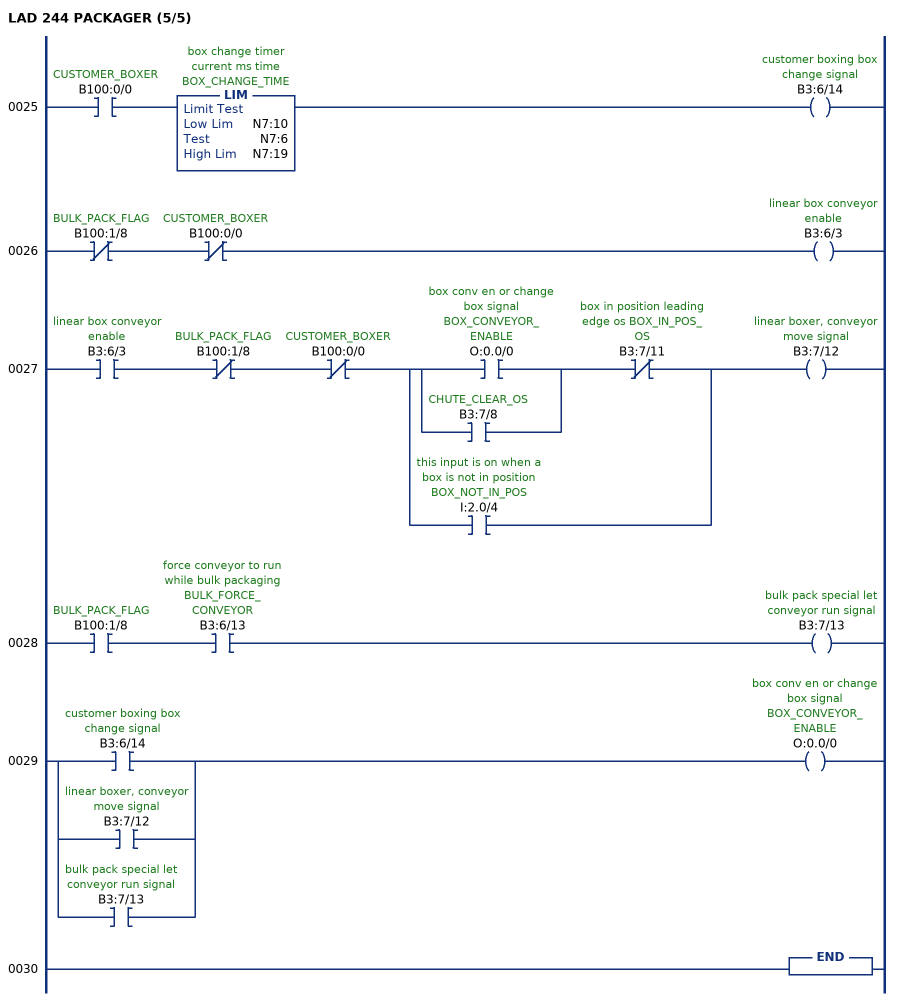
% Rung: 25 %
SOR XIC B100:0/0 LIM N7:10 N7:6 N7:19 OTE B3:6/14 EOR
%   B100:0/0  CUSTOMER_BOXER %
%   N7:10  CHUTE_CLOSED_TIME  "time at which chute door is considered closed" %
%   N7:6  BOX_CHANGE_TIME  "box change timer current ms time" %
%   N7:19  "end of customer boxer, box change signal" %
%   B3:6/14  "customer boxing box change signal" %
% Rung: 26 %
SOR XIO B100:1/8 XIO B100:0/0 OTE B3:6/3 EOR
%   B100:1/8  BULK_PACK_FLAG %
%   B100:0/0  CUSTOMER_BOXER %
%   B3:6/3  "linear box conveyor enable" %
% Rung: 27 %
SOR XIC B3:6/3 XIO B100:1/8 XIO B100:0/0 BST BST XIC O:0.0/0 NXB XIC B3:7/8 BND XIO B3:7/11 NXB XIC I:2.0/4 BND OTE B3:7/12 EOR
%   B3:6/3  "linear box conveyor enable" %
%   B100:1/8  BULK_PACK_FLAG %
%   B100:0/0  CUSTOMER_BOXER %
%   O:0.0/0  BOX_CONVEYOR_ENABLE  "box conv en or change box signal" %
%   B3:7/8  CHUTE_CLEAR_OS %
%   B3:7/11  BOX_IN_POS_OS  "box in position leading edge os" %
%   I:2.0/4  BOX_NOT_IN_POS  "this input is on when a box is not in position" %
%   B3:7/12  "linear boxer, conveyor move signal" %
% Rung: 28 %
SOR XIC B100:1/8 XIC B3:6/13 OTE B3:7/13 EOR
%   B100:1/8  BULK_PACK_FLAG %
%   B3:6/13  BULK_FORCE_CONVEYOR  "force conveyor to run while bulk packaging" %
%   B3:7/13  "bulk pack special let conveyor run signal" %
% Rung: 29 %
SOR BST XIC B3:6/14 NXB XIC B3:7/12 NXB XIC B3:7/13 BND OTE O:0.0/0 EOR
%   B3:6/14  "customer boxing box change signal" %
%   B3:7/12  "linear boxer, conveyor move signal" %
%   B3:7/13  "bulk pack special let conveyor run signal" %
%   O:0.0/0  BOX_CONVEYOR_ENABLE  "box conv en or change box signal" %
% Rung: 30 %
SOR END EOR

LADDER 245 "NO PACKAGE"
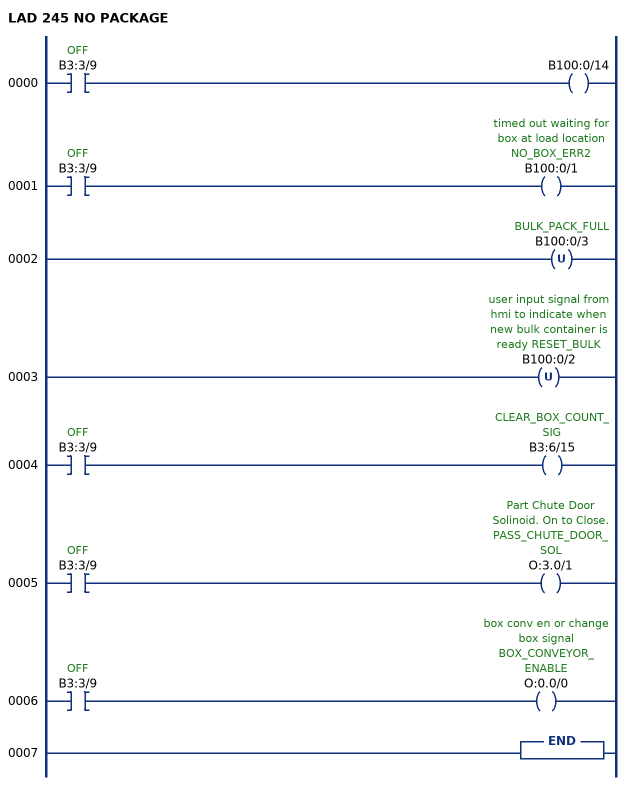
% Rung: 0 %
SOR XIC B3:3/9 OTE B100:0/14 EOR
%   B3:3/9  OFF %
% Rung: 1 %
SOR XIC B3:3/9 OTE B100:0/1 EOR
%   B3:3/9  OFF %
%   B100:0/1  NO_BOX_ERR2  "timed out waiting for box at load location" %
% Rung: 2 %
SOR OTU B100:0/3 EOR
%   B100:0/3  BULK_PACK_FULL %
% Rung: 3 %
SOR OTU B100:0/2 EOR
%   B100:0/2  RESET_BULK  "user input signal from hmi to indicate when new bulk container is ready" %
% Rung: 4 %
SOR XIC B3:3/9 OTE B3:6/15 EOR
%   B3:3/9  OFF %
%   B3:6/15  CLEAR_BOX_COUNT_SIG %
% Rung: 5 %
SOR XIC B3:3/9 OTE O:3.0/1 EOR
%   B3:3/9  OFF %
%   O:3.0/1  PASS_CHUTE_DOOR_SOL  "Part Chute Door Solinoid. On to Close." %
% Rung: 6 %
SOR XIC B3:3/9 OTE O:0.0/0 EOR
%   B3:3/9  OFF %
%   O:0.0/0  BOX_CONVEYOR_ENABLE  "box conv en or change box signal" %
% Rung: 7 %
SOR END EOR

LADDER 246 "RATE1"
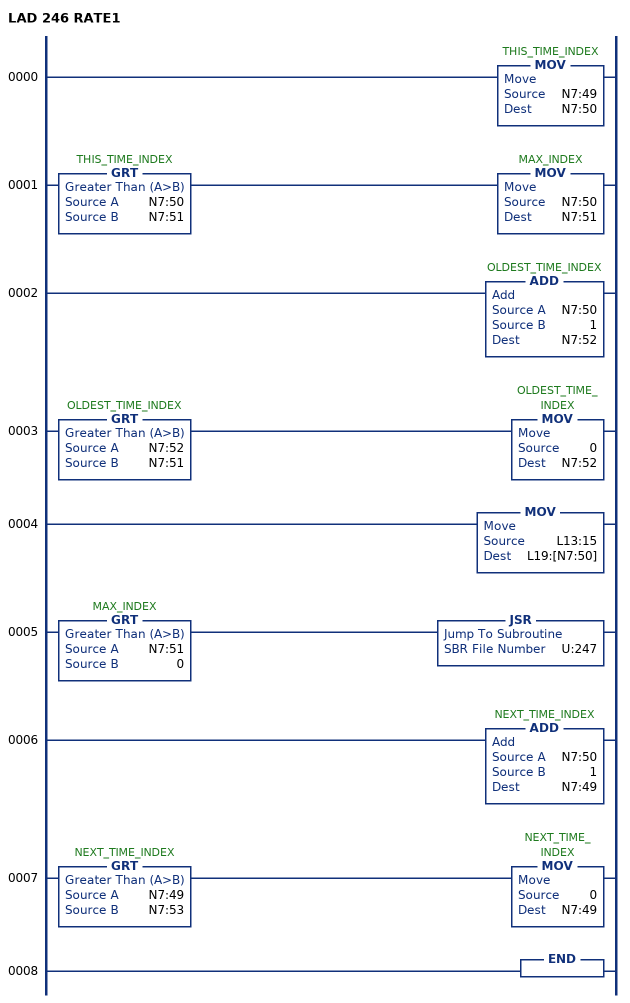
% Rung: 0 %
SOR MOV N7:49 N7:50 EOR
%   N7:49  NEXT_TIME_INDEX %
%   N7:50  THIS_TIME_INDEX %
% Rung: 1 %
SOR GRT N7:50 N7:51 MOV N7:50 N7:51 EOR
%   N7:50  THIS_TIME_INDEX %
%   N7:51  MAX_INDEX %
% Rung: 2 %
SOR ADD N7:50 1 N7:52 EOR
%   N7:50  THIS_TIME_INDEX %
%   N7:52  OLDEST_TIME_INDEX %
% Rung: 3 %
SOR GRT N7:52 N7:51 MOV 0 N7:52 EOR
%   N7:52  OLDEST_TIME_INDEX %
%   N7:51  MAX_INDEX %
% Rung: 4 %
SOR MOV L13:15 L19:[N7:50] EOR
%   L13:15  THE_TIME %
%   N7:50  THIS_TIME_INDEX %
% Rung: 5 %
SOR GRT N7:51 0 JSR U:247 EOR
%   N7:51  MAX_INDEX %
% Rung: 6 %
SOR ADD N7:50 1 N7:49 EOR
%   N7:50  THIS_TIME_INDEX %
%   N7:49  NEXT_TIME_INDEX %
% Rung: 7 %
SOR GRT N7:49 N7:53 MOV 0 N7:49 EOR
%   N7:49  NEXT_TIME_INDEX %
%   N7:53  UPPER_INDEX_LIMIT %
% Rung: 8 %
SOR END EOR

LADDER 247 "RATE2"
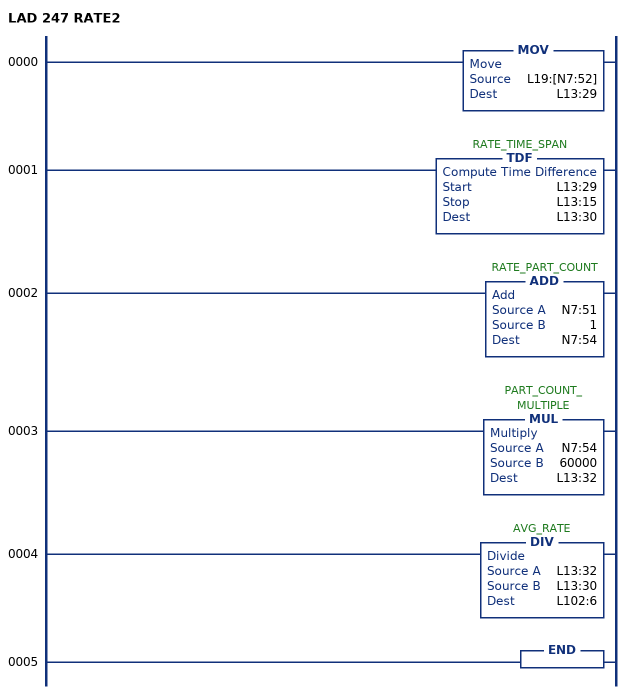
% Rung: 0 %
SOR MOV L19:[N7:52] L13:29 EOR
%   N7:52  OLDEST_TIME_INDEX %
% Rung: 1 %
SOR TDF L13:29 L13:15 L13:30 EOR
%   L13:15  THE_TIME %
%   L13:30  RATE_TIME_SPAN %
% Rung: 2 %
SOR ADD N7:51 1 N7:54 EOR
%   N7:51  MAX_INDEX %
%   N7:54  RATE_PART_COUNT %
% Rung: 3 %
SOR MUL N7:54 60000 L13:32 EOR
%   N7:54  RATE_PART_COUNT %
%   L13:32  PART_COUNT_MULTIPLE %
% Rung: 4 %
SOR DIV L13:32 L13:30 L102:6 EOR
%   L13:32  PART_COUNT_MULTIPLE %
%   L13:30  RATE_TIME_SPAN %
%   L102:6  AVG_RATE %
% Rung: 5 %
SOR END EOR

LADDER 248 "RESET RATE"
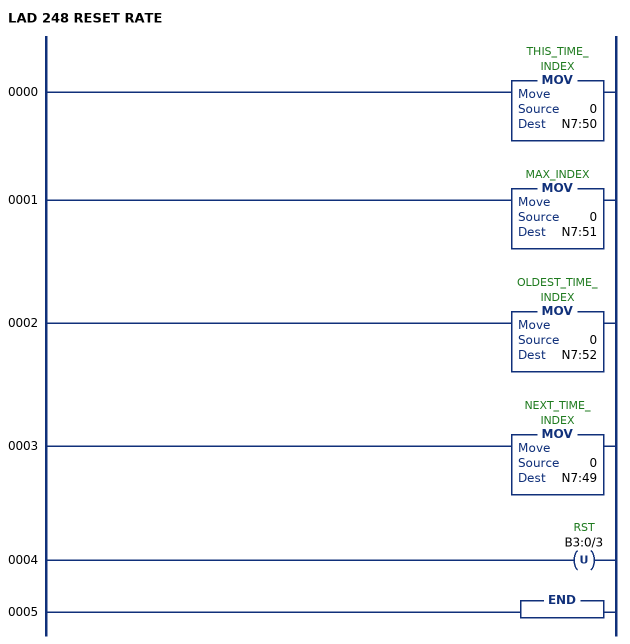
% Rung: 0 %
SOR MOV 0 N7:50 EOR
%   N7:50  THIS_TIME_INDEX %
% Rung: 1 %
SOR MOV 0 N7:51 EOR
%   N7:51  MAX_INDEX %
% Rung: 2 %
SOR MOV 0 N7:52 EOR
%   N7:52  OLDEST_TIME_INDEX %
% Rung: 3 %
SOR MOV 0 N7:49 EOR
%   N7:49  NEXT_TIME_INDEX %
% Rung: 4 %
SOR OTU B3:0/3 EOR
%   B3:0/3  RST %
% Rung: 5 %
SOR END EOR

LADDER 249 "NP STOP"    % stop on no good %
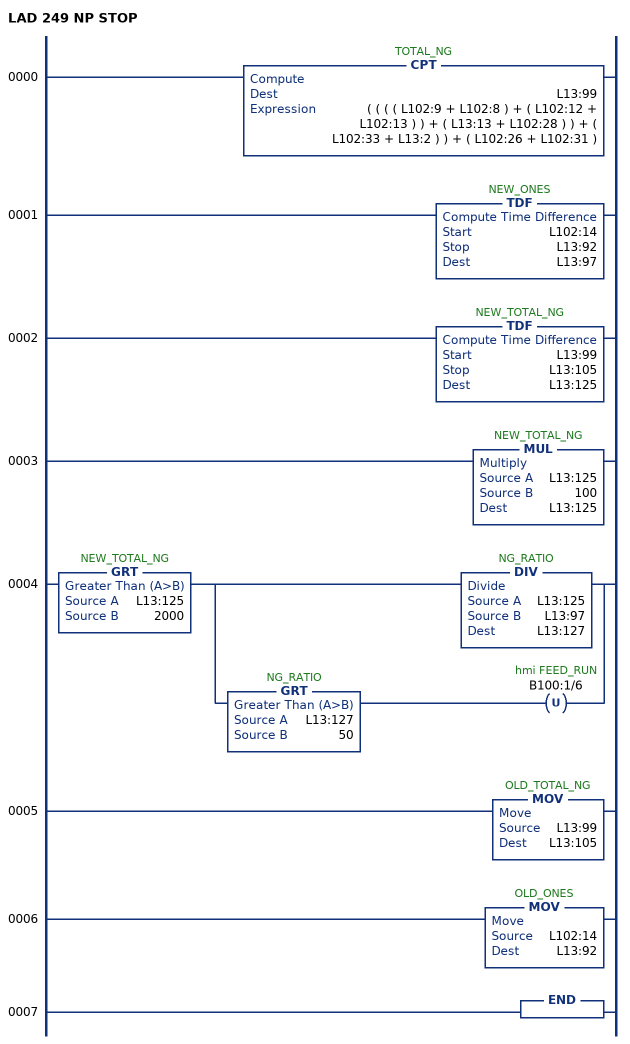
% Rung: 0 %
SOR CPT L13:99 " ( ( ( ( L102:9 + L102:8 ) + ( L102:12 + L102:13 ) ) + ( L13:13 + L102:28 ) ) + ( L102:33 + L13:2 ) ) + ( L102:26 + L102:31 ) " EOR
%   L13:99  TOTAL_NG %
%   L102:9  "too wide bottom" %
%   L102:8  "too close bottom" %
%   L102:12  "too close top count" %
%   L102:13  "too wide top count" %
%   L102:28  I1_I5_SKIPPEDCOUNT %
%   L102:33  I2_I6_SKIPPEDCOUNT %
%   L102:26  I1_I5_FAIL_COUNT %
%   L102:31  I2_I6_FAIL_COUNT %
% Rung: 1 %
SOR TDF L102:14 L13:92 L13:97 EOR
%   L102:14  ONES %
%   L13:92  OLD_ONES %
%   L13:97  NEW_ONES %
% Rung: 2 %
SOR TDF L13:99 L13:105 L13:125 EOR
%   L13:99  TOTAL_NG %
%   L13:105  OLD_TOTAL_NG %
%   L13:125  NEW_TOTAL_NG %
% Rung: 3 %
SOR MUL L13:125 100 L13:125 EOR
%   L13:125  NEW_TOTAL_NG %
% Rung: 4 %
SOR GRT L13:125 2000 BST DIV L13:125 L13:97 L13:127 NXB GRT L13:127 50 OTU B100:1/6 BND EOR
%   L13:125  NEW_TOTAL_NG %
%   L13:97  NEW_ONES %
%   L13:127  NG_RATIO %
%   B100:1/6  FEED_RUN  "hmi" %
% Rung: 5 %
SOR MOV L13:99 L13:105 EOR
%   L13:99  TOTAL_NG %
%   L13:105  OLD_TOTAL_NG %
% Rung: 6 %
SOR MOV L102:14 L13:92 EOR
%   L102:14  ONES %
%   L13:92  OLD_ONES %
% Rung: 7 %
SOR END EOR

LADDER 250 "SPEED BOT"    % high speed %
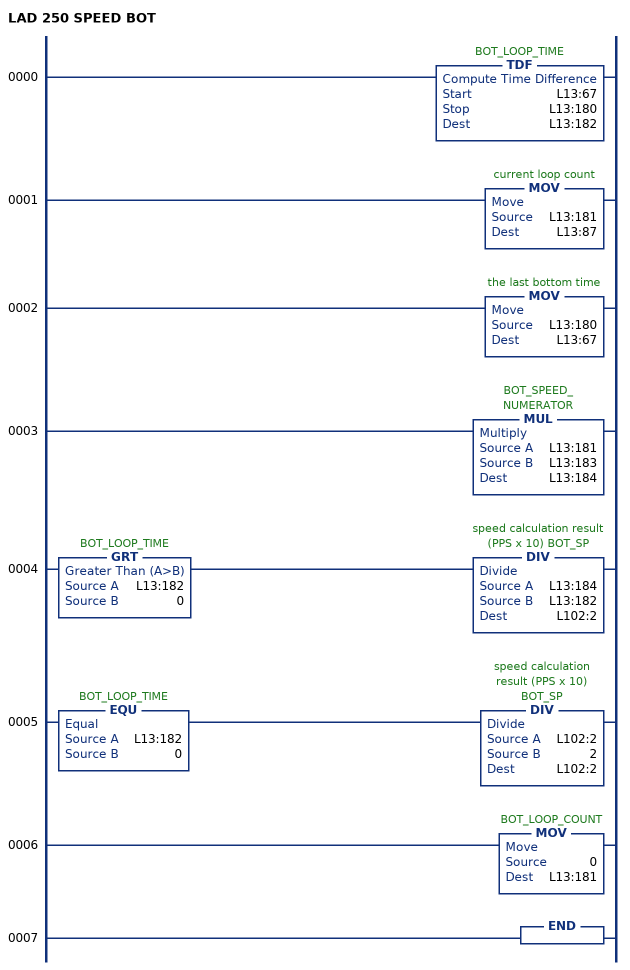
% Rung: 0 %
SOR TDF L13:67 L13:180 L13:182 EOR
%   L13:67  "the last bottom time" %
%   L13:180  BOT_THIS_TIME  "rtc bot belt movement event time" %
%   L13:182  BOT_LOOP_TIME %
% Rung: 1 %
SOR MOV L13:181 L13:87 EOR
%   L13:181  BOT_LOOP_COUNT %
%   L13:87  "current loop count" %
% Rung: 2 %
SOR MOV L13:180 L13:67 EOR
%   L13:180  BOT_THIS_TIME  "rtc bot belt movement event time" %
%   L13:67  "the last bottom time" %
% Rung: 3 %
SOR MUL L13:181 L13:183 L13:184 EOR
%   L13:181  BOT_LOOP_COUNT %
%   L13:183  TKS_PER_SECOND %
%   L13:184  BOT_SPEED_NUMERATOR %
% Rung: 4 %
SOR GRT L13:182 0 DIV L13:184 L13:182 L102:2 EOR
%   L13:182  BOT_LOOP_TIME %
%   L13:184  BOT_SPEED_NUMERATOR %
%   L102:2  BOT_SP  "speed calculation result (PPS x 10)" %
% Rung: 5 %
SOR EQU L13:182 0 DIV L102:2 2 L102:2 EOR
%   L13:182  BOT_LOOP_TIME %
%   L102:2  BOT_SP  "speed calculation result (PPS x 10)" %
% Rung: 6 %
SOR MOV 0 L13:181 EOR
%   L13:181  BOT_LOOP_COUNT %
% Rung: 7 %
SOR END EOR

LADDER 251 "SPEED TOP"    % high speed %
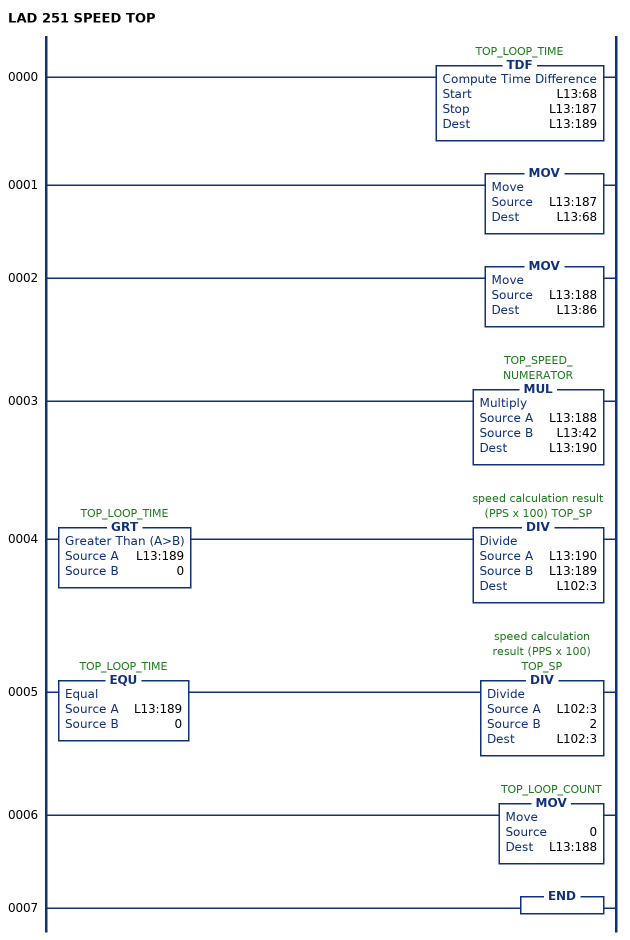
% Rung: 0 %
SOR TDF L13:68 L13:187 L13:189 EOR
%   L13:187  TOP_THIS_TIME  "rtc top belt movement event time" %
%   L13:189  TOP_LOOP_TIME %
% Rung: 1 %
SOR MOV L13:187 L13:68 EOR
%   L13:187  TOP_THIS_TIME  "rtc top belt movement event time" %
% Rung: 2 %
SOR MOV L13:188 L13:86 EOR
%   L13:188  TOP_LOOP_COUNT %
% Rung: 3 %
SOR MUL L13:188 L13:42 L13:190 EOR
%   L13:188  TOP_LOOP_COUNT %
%   L13:190  TOP_SPEED_NUMERATOR %
% Rung: 4 %
SOR GRT L13:189 0 DIV L13:190 L13:189 L102:3 EOR
%   L13:189  TOP_LOOP_TIME %
%   L13:190  TOP_SPEED_NUMERATOR %
%   L102:3  TOP_SP  "speed calculation result (PPS x 100)" %
% Rung: 5 %
SOR EQU L13:189 0 DIV L102:3 2 L102:3 EOR
%   L13:189  TOP_LOOP_TIME %
%   L102:3  TOP_SP  "speed calculation result (PPS x 100)" %
% Rung: 6 %
SOR MOV 0 L13:188 EOR
%   L13:188  TOP_LOOP_COUNT %
% Rung: 7 %
SOR END EOR

LADDER 252 "P BOT"    % high speed %
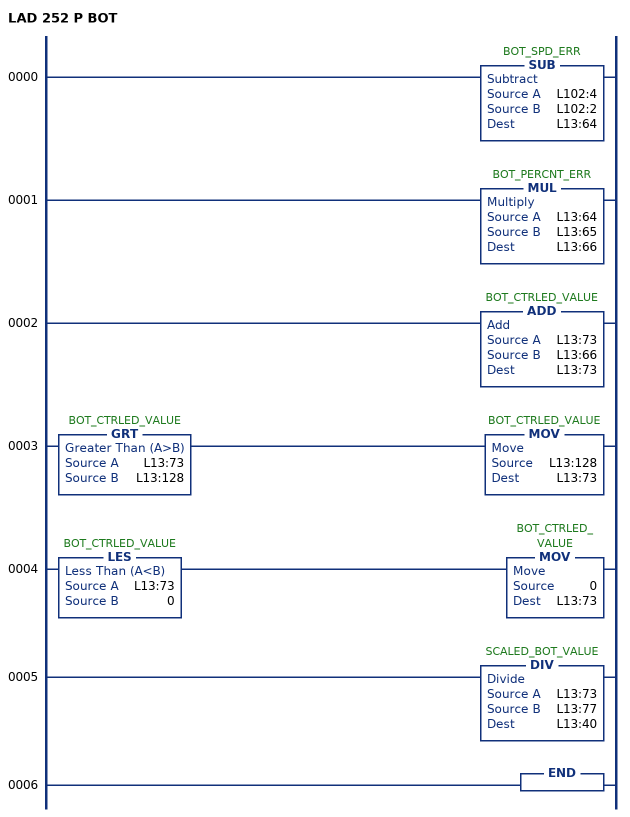
% Rung: 0 %
SOR SUB L102:4 L102:2 L13:64 EOR
%   L102:4  BOT_SPD_SETPOINT %
%   L102:2  BOT_SP  "speed calculation result (PPS x 10)" %
%   L13:64  BOT_SPD_ERR %
% Rung: 1 %
SOR MUL L13:64 L13:65 L13:66 EOR
%   L13:64  BOT_SPD_ERR %
%   L13:65  POS5SHIFT %
%   L13:66  BOT_PERCNT_ERR %
% Rung: 2 %
SOR ADD L13:73 L13:66 L13:73 EOR
%   L13:73  BOT_CTRLED_VALUE %
%   L13:66  BOT_PERCNT_ERR %
% Rung: 3 %
SOR GRT L13:73 L13:128 MOV L13:128 L13:73 EOR
%   L13:73  BOT_CTRLED_VALUE %
%   L13:128  "how much top has shifted since measurment" %
% Rung: 4 %
SOR LES L13:73 0 MOV 0 L13:73 EOR
%   L13:73  BOT_CTRLED_VALUE %
% Rung: 5 %
SOR DIV L13:73 L13:77 L13:40 EOR
%   L13:73  BOT_CTRLED_VALUE %
%   L13:40  SCALED_BOT_VALUE %
% Rung: 6 %
SOR END EOR

LADDER 253 "P TOP"    % high speed %
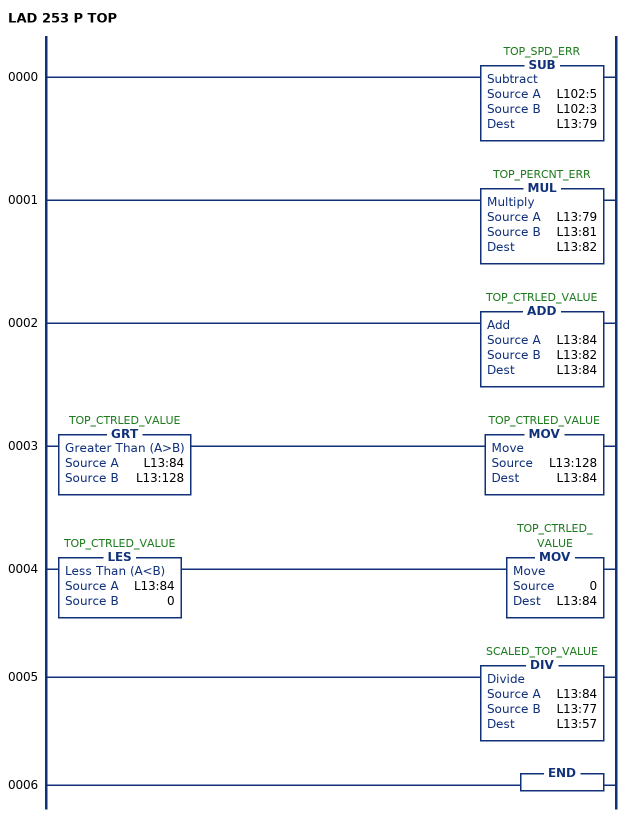
% Rung: 0 %
SOR SUB L102:5 L102:3 L13:79 EOR
%   L102:5  TOP_SPD_SETPOINT %
%   L102:3  TOP_SP  "speed calculation result (PPS x 100)" %
%   L13:79  TOP_SPD_ERR %
% Rung: 1 %
SOR MUL L13:79 L13:81 L13:82 EOR
%   L13:79  TOP_SPD_ERR %
%   L13:81  TOP_FDBK_RATIO %
%   L13:82  TOP_PERCNT_ERR %
% Rung: 2 %
SOR ADD L13:84 L13:82 L13:84 EOR
%   L13:84  TOP_CTRLED_VALUE %
%   L13:82  TOP_PERCNT_ERR %
% Rung: 3 %
SOR GRT L13:84 L13:128 MOV L13:128 L13:84 EOR
%   L13:84  TOP_CTRLED_VALUE %
%   L13:128  "how much top has shifted since measurment" %
% Rung: 4 %
SOR LES L13:84 0 MOV 0 L13:84 EOR
%   L13:84  TOP_CTRLED_VALUE %
% Rung: 5 %
SOR DIV L13:84 L13:77 L13:57 EOR
%   L13:84  TOP_CTRLED_VALUE %
%   L13:57  SCALED_TOP_VALUE %
% Rung: 6 %
SOR END EOR

LADDER 254 "TOTALCOUNT"
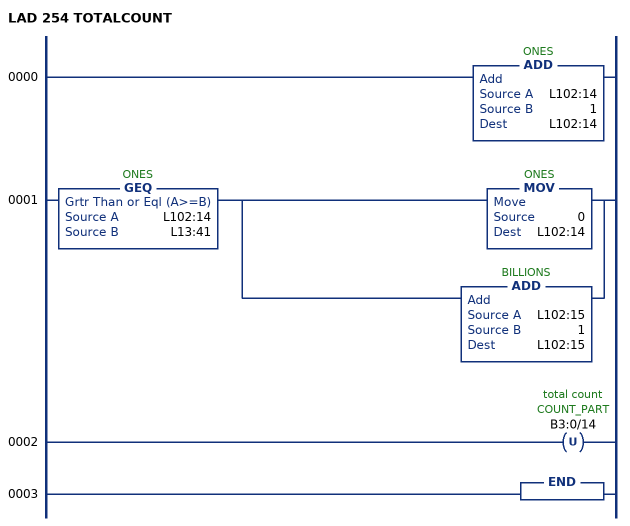
% Rung: 0 %
SOR ADD L102:14 1 L102:14 EOR
%   L102:14  ONES %
% Rung: 1 %
SOR GEQ L102:14 L13:41 BST MOV 0 L102:14 NXB ADD L102:15 1 L102:15 BND EOR
%   L102:14  ONES %
%   L13:41  "skipped count change in the last 3 seconds" %
%   L102:15  BILLIONS %
% Rung: 2 %
SOR OTU B3:0/14 EOR
%   B3:0/14  COUNT_PART  "total count" %
% Rung: 3 %
SOR END EOR

LADDER 255 "SAVED"
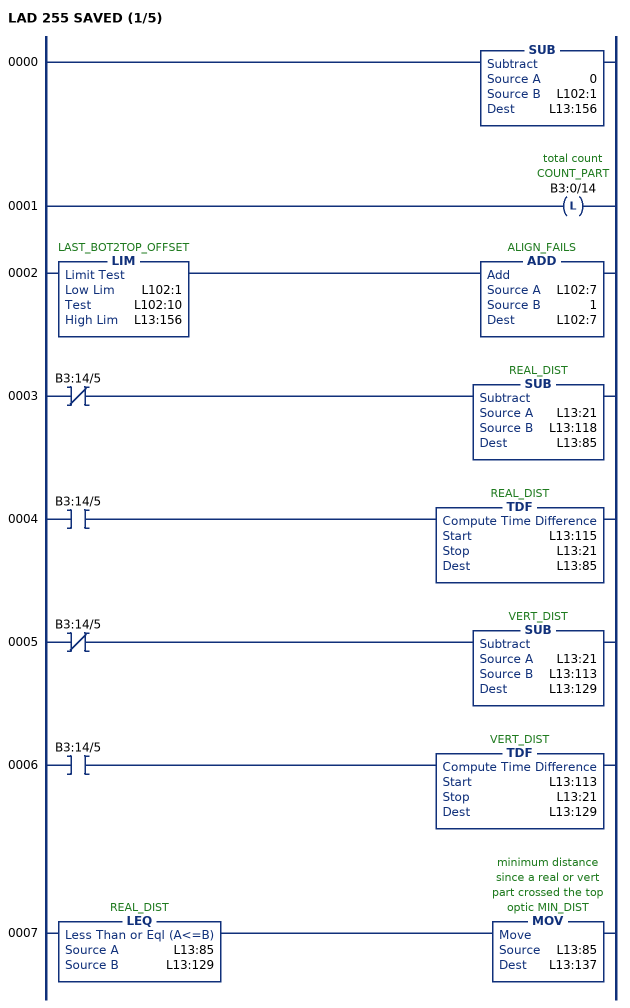
% Rung: 0 %
SOR SUB 0 L102:1 L13:156 EOR
%   L102:1  MAX_OFFSET  "transition zone width" %
% Rung: 1 %
SOR OTL B3:0/14 EOR
%   B3:0/14  COUNT_PART  "total count" %
% Rung: 2 %
SOR LIM L102:1 L102:10 L13:156 ADD L102:7 1 L102:7 EOR
%   L102:1  MAX_OFFSET  "transition zone width" %
%   L102:10  LAST_BOT2TOP_OFFSET %
%   L102:7  ALIGN_FAILS %
% Rung: 3 %
SOR XIO B3:14/5 SUB L13:21 L13:118 L13:85 EOR
%   L13:21  TOP_POSITION %
%   L13:118  REAL_CL_POSITION  "real part center line in raw position" %
%   L13:85  REAL_DIST %
% Rung: 4 %
SOR XIC B3:14/5 TDF L13:115 L13:21 L13:85 EOR
%   L13:115  TRAILING_EDGE_POS  "top optic trailing edge position" %
%   L13:21  TOP_POSITION %
%   L13:85  REAL_DIST %
% Rung: 5 %
SOR XIO B3:14/5 SUB L13:21 L13:113 L13:129 EOR
%   L13:21  TOP_POSITION %
%   L13:113  VIRT_CL_POSITION  "virtual part center line transfer from the bottom in raw position" %
%   L13:129  VERT_DIST %
% Rung: 6 %
SOR XIC B3:14/5 TDF L13:113 L13:21 L13:129 EOR
%   L13:113  VIRT_CL_POSITION  "virtual part center line transfer from the bottom in raw position" %
%   L13:21  TOP_POSITION %
%   L13:129  VERT_DIST %
% Rung: 7 %
SOR LEQ L13:85 L13:129 MOV L13:85 L13:137 EOR
%   L13:85  REAL_DIST %
%   L13:129  VERT_DIST %
%   L13:137  MIN_DIST  "minimum distance since a real or vert part crossed the top optic" %

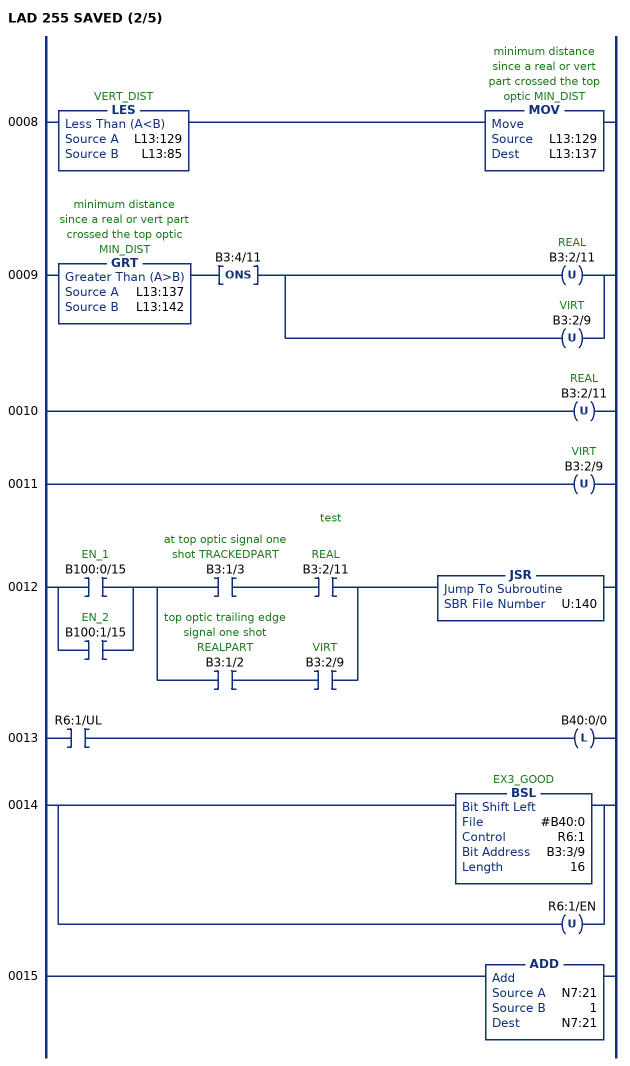
% Rung: 8 %
SOR LES L13:129 L13:85 MOV L13:129 L13:137 EOR
%   L13:129  VERT_DIST %
%   L13:85  REAL_DIST %
%   L13:137  MIN_DIST  "minimum distance since a real or vert part crossed the top optic" %
% Rung: 9 %
SOR GRT L13:137 L13:142 ONS B3:4/11 BST OTU B3:2/11 NXB OTU B3:2/9 BND EOR
%   L13:137  MIN_DIST  "minimum distance since a real or vert part crossed the top optic" %
%   L13:142  LAST_ALIGNMENT_FAILS %
%   B3:2/11  REAL %
%   B3:2/9  VIRT %
% Rung: 10 %
SOR OTU B3:2/11 EOR
%   B3:2/11  REAL %
% Rung: 11 %
SOR OTU B3:2/9 EOR
%   B3:2/9  VIRT %
% Rung: 12 %
% test %
SOR BST XIC B100:0/15 NXB XIC B100:1/15 BND BST XIC B3:1/3 XIC B3:2/11 NXB XIC B3:1/2 XIC B3:2/9 BND JSR U:140 EOR
%   B100:0/15  EN_1 %
%   B100:1/15  EN_2 %
%   B3:1/3  TRACKEDPART  "at top optic signal one shot" %
%   B3:2/11  REAL %
%   B3:1/2  REALPART  "top optic trailing edge signal one shot" %
%   B3:2/9  VIRT %
% Rung: 13 %
SOR XIC R6:1/UL OTL B40:0/0 EOR
% Rung: 14 %
SOR BST BSL #B40:0 R6:1 B3:3/9 16 NXB OTU R6:1/EN BND EOR
%   B40:0  EX3_GOOD %
%   B3:3/9  OFF %
% Rung: 15 %
SOR ADD N7:21 1 N7:21 EOR

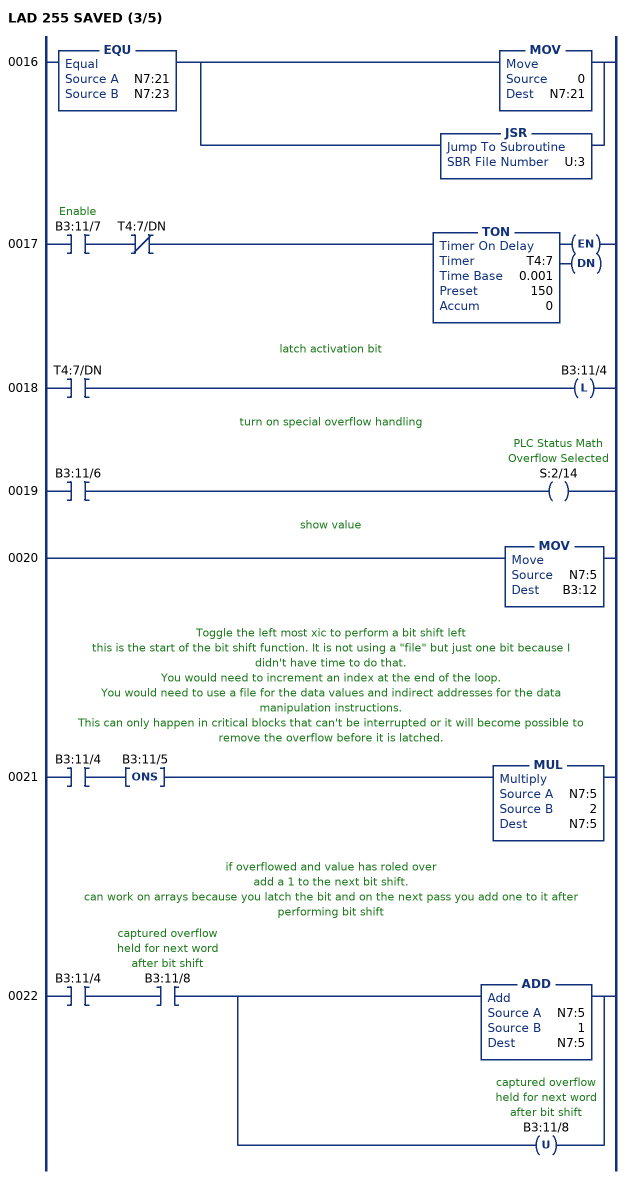
% Rung: 16 %
SOR EQU N7:21 N7:23 BST MOV 0 N7:21 NXB JSR U:3 BND EOR
% Rung: 17 %
SOR XIC B3:11/7 XIO T4:7/DN TON T4:7 0.001 150 0 EOR
%   B3:11/7  "Enable" %
% Rung: 18 %
% latch activation bit %
SOR XIC T4:7/DN OTL B3:11/4 EOR
% Rung: 19 %
% turn on special overflow handling %
SOR XIC B3:11/6 OTE S:2/14 EOR
%   S:2/14  "PLC Status Math Overflow Selected" %
% Rung: 20 %
% show value %
SOR MOV N7:5 B3:12 EOR
% Rung: 21 %
% Toggle the left most xic to perform a bit shift left
% 
% this is the start of the bit shift function. It is not using a "file" but just one bit because I didn't have time to do that.
% You would need to increment an index at the end of the loop.
% You would need to use a file for the data values and indirect addresses for the data manipulation instructions.
% 
% This can only happen in critical blocks that can't be interrupted or it will become possible to remove the overflow before it is latched. %
SOR XIC B3:11/4 ONS B3:11/5 MUL N7:5 2 N7:5 EOR
% Rung: 22 %
% if overflowed and value has roled over
% add a 1 to the next bit shift.
% can work on arrays because you latch the bit and on the next pass you add one to it after performing bit shift %
SOR XIC B3:11/4 XIC B3:11/8 BST ADD N7:5 1 N7:5 NXB OTU B3:11/8 BND EOR
%   B3:11/8  "captured overflow held for next word after bit shift" %

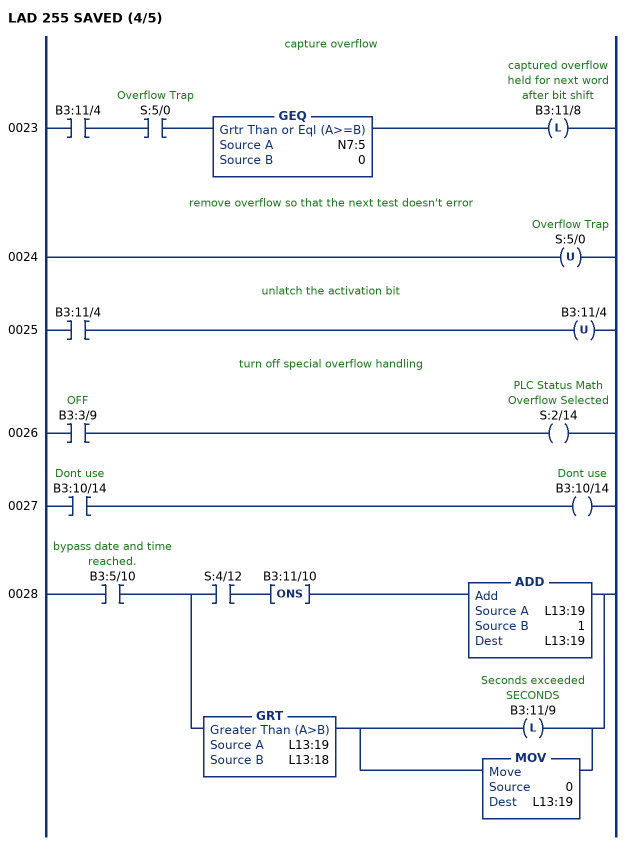
% Rung: 23 %
% capture overflow %
SOR XIC B3:11/4 XIC S:5/0 GEQ N7:5 0 OTL B3:11/8 EOR
%   S:5/0  "Overflow Trap" %
%   B3:11/8  "captured overflow held for next word after bit shift" %
% Rung: 24 %
% remove overflow so that the next test doesn't error %
SOR OTU S:5/0 EOR
%   S:5/0  "Overflow Trap" %
% Rung: 25 %
% unlatch the activation bit %
SOR XIC B3:11/4 OTU B3:11/4 EOR
% Rung: 26 %
% turn off special overflow handling %
SOR XIC B3:3/9 OTE S:2/14 EOR
%   B3:3/9  OFF %
%   S:2/14  "PLC Status Math Overflow Selected" %
% Rung: 27 %
SOR XIC B3:10/14 OTE B3:10/14 EOR
%   B3:10/14  "Dont use" %
% Rung: 28 %
SOR XIC B3:5/10 BST XIC S:4/12 ONS B3:11/10 ADD L13:19 1 L13:19 NXB GRT L13:19 L13:18 BST OTL B3:11/9 NXB MOV 0 L13:19 BND BND EOR
%   B3:5/10  "bypass date and time reached." %
%   L13:18  MAX %
%   B3:11/9  SECONDS  "Seconds exceeded" %

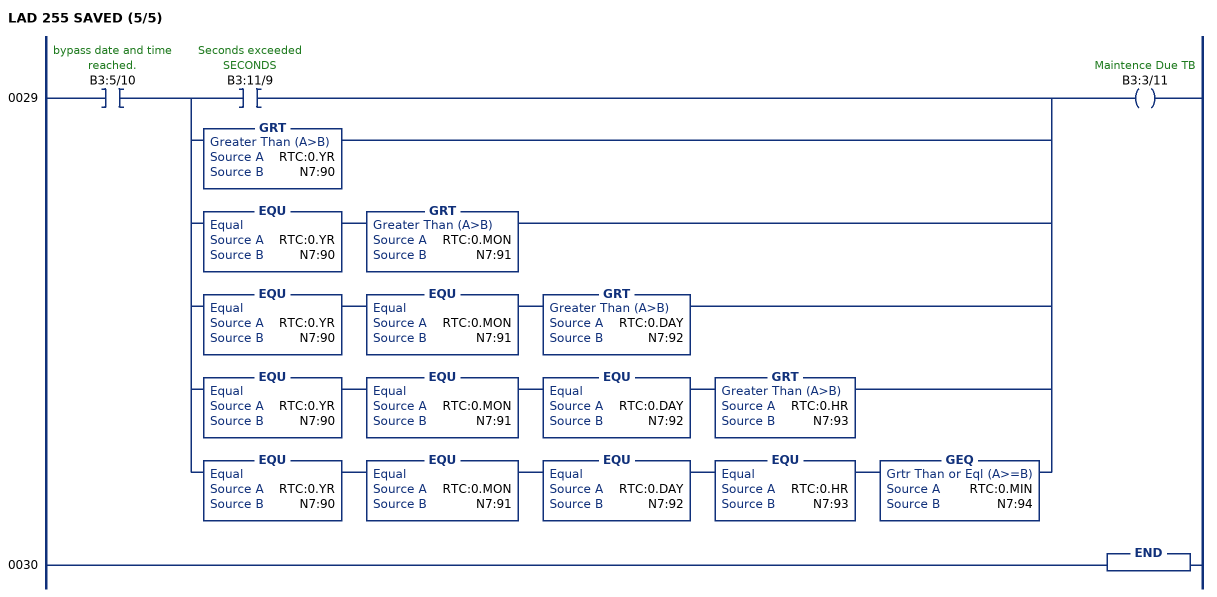
% Rung: 29 %
SOR XIC B3:5/10 BST XIC B3:11/9 NXB GRT RTC:0.YR N7:90 NXB EQU RTC:0.YR N7:90 GRT RTC:0.MON N7:91 NXB EQU RTC:0.YR N7:90 EQU RTC:0.MON N7:91 GRT RTC:0.DAY N7:92 NXB EQU RTC:0.YR N7:90 EQU RTC:0.MON N7:91 EQU RTC:0.DAY N7:92 GRT RTC:0.HR N7:93 NXB EQU RTC:0.YR N7:90 EQU RTC:0.MON N7:91 EQU RTC:0.DAY N7:92 EQU RTC:0.HR N7:93 GEQ RTC:0.MIN N7:94 BND OTE B3:3/11 EOR
%   B3:5/10  "bypass date and time reached." %
%   B3:11/9  SECONDS  "Seconds exceeded" %
%   N7:90  RTC %
%   B3:3/11  TB  "Maintence Due" %
% Rung: 30 %
SOR END EOR

OTHER DOCUMENTED ADDRESSES
  B38:0  EX1_GOOD
  B189:0/0  "change box"
  B189:0/9  "override boxing ok or not full signal"
  B189:0/11  "HMI force door close"
  B196:1/0  "Chute door is closed"
  B196:1/1  "control chute door"
  B196:1/13  "force box conveyor on"
  B196:3/0  "for hmi to continue production unlatched by hmi"
  HSC:0.0  "top"
  HSC:0.3/6  "Underflow interrupt"
  HSC:0.3/7  "Overflow interrupt"
  HSC:1.0  "bot"
  HSC:1.3/6  "Underflow interrupt"
  HSC:1.3/7  "Overflow interrupt"
  I7_TRAC  
  I:0.0/0  "Encoder Signal "A""
  I:0.0/1  "Encoder Signal "B""
  I:0.0/4  "Encoder Signal "A""
  I:0.0/5  "Encoder Signal "B""
  I:0.1/4  "not used"
  I:0.1/5  "not used"
  I:0.1/6  "not used"
  I:0.1/7  "not used"
  I:0.1/8  "not used"
  I:0.1/9  "not used"
  I:0.1/10  "not used"
  I:0.1/11  "not used"
  I:0.1/12  "not used"
  I:0.1/13  "not used"
  I:0.1/14  "not used"
  I:0.1/15  "not used"
  I:0.2  "not used"
  I:0.2/3  "Packaging Conveyor full"
  I:0.2/4  "Packaging Conveyor Box in Position"
  I:0.3  "not used"
  I:0.4  "Spare Analog Input 1"
  I:0.5  "Spare Analog Input 2"
  I:0.6  "Spare Analog Input 3"
  I:2.0/0  FRONT_ESTOP
  I:2.0/1  REAR_ESTOP
  I:2.0/8  FRONT_DOOR  "front door signal ce models only"
  I:2.0/9  REAR_DOOR  "rear door signal ce models only"
  I:2.0/11  "spare"
  L13:132  "set speed"
  L13:133  "controlled speed"
  L23:19  TOP_OPT_FAIL_CT
  L23:34  AIR_PRESSURE_FAULT
  L28:0  INS_1_TIME
  L29:0  INS_1_POS
  L30:0  INS_5_TIME
  L31:0  INS_5_POS
  L32:0  INS_6_TIME
  L33:0  INS_6_POS
  L192:1  BOT_LAST_TIME  "rtc bot belt previous movement event time"
  L192:2  BOT_CYCLE_TIME  "rtc bot belt time between events"
  L192:7  FROM_REAL  "distance from real part signal at optic location"
  L192:8  FROM_TRACKED  "distance from tracked part signal at optic location"
  L192:16  TOP_LAST_TIME  "rtc top belt previous movement event time"
  L192:17  TOP_CYCLE_TIME  "rtc top belt time between events"
  L199:5  ACQTM51
  L199:6  ACQTM52
  L199:7  ACQTM53
  L199:9  "ones"
  L199:10  "billions"
  L199:13  DUMP_LONG
  L199:15  ACQTM11
  L199:16  ACQTM12
  L199:17  ACQTM13
  L199:20  RESULTTM1
  L199:22  CLEARTIME5COUNT
  L199:23  CLEARTIME6COUNT
  L199:24  ACQTM61
  L199:25  ACQTM62
  L199:26  ACQTM63
  L199:27  TMSINCETRIG1
  L199:29  TMSINCETRIG5
  L199:30  TMSINCETRIG6
  L199:31  CLEARTIME1COUNT
  L199:32  RESULTTM5
  L199:33  RESULTTM6
  L199:34  MAXACQTM1
  L199:36  MAXACQTM6
  N7  
  N101:2  I3_TRIG_LOC
  N101:3  I4_TRIG_LOC
  O:0.0/1  "spare"
  O:0.0/11  "Spare"
  O:0.0/12  "not used"
  O:0.0/13  "not used"
  O:0.0/14  "not used"
  O:0.0/15  "not used"
  O:0.1  "not used"
  O:0.2  "not used"
  O:0.3  "not used"
  O:0.5  "spare analog output"
  O:3.0/0  "spare"
  O:3.0/2  "spare"
  O:3.0/3  "light curtain range selection /* needed? */"
  O:3.0/7  "door unlocks on CE models"
  O:3.0/8  "Light?"
  O:3.0/9  NUT_HOPPER  "Nut Hopper Enable"
  O:3.0/11  NUT_FEEDER_AIR  "Nut Feeder Bowl Air Enable"
  PFILE:6  "check for part jams"
  PFILE:10  "Bottom belt HSC"
  PFILE:12  "Top belt HSC"
  Q2:55  END_OF_MAIN
  Q5:94  END_OF_BELTS
  T20:0  "Trigger On Time"
  U:9  "slow data"
  U:24  "check skipped fail rate"
  U:28  "faults"
  U:29  "speed"
  U:30  "count"
  U:31  "rate calc"
  U:32  "boxer"
  U:33  "bulk pack"
  U:34  "customer boxing unit signals"
  U:35  "cleanup"

COMMENTS NOT ATTACHED TO A CURRENT RUNG
  R6:2: B41 is the top good 3 file
  R6:6/DN: B35 is the top NG file
  R6:10/DN: B37 is the top good 1 file
  R6:11/DN: B39 is the top good 2 file
  B100:1/15: what is this code for?
  R6:0: B36 is the bottom GOOD file
  R6:10: B37 is the top good 1 file
  R6:6: B35 is the top NG file
  R6:4: B34 is the bottom NG file

REVISION NOTES
  13: updated count reset
  14: added io moduals
  15: multiple steps toward new hmi integration
  21: test
  27: fix error if bulk pack and no boxing fallout were on

DATA TABLE (non-zero values as saved)
DATA B3
% B3:0 % 0X8802 0X1160 0X4041 0X9101 0XCCAF 0X1514 0X0438 0X0461 0X2F80 0X22DC
% B3:10 % 0X21F8 0X40C6 0X4000 0X134C 0X0001 0X0000 0X0000 0X0000 0X0000 0X0000
% B3:50 % 0X0001 0X0000 0X0000 0X0000 0X0000 0X0000 0X0000 0X0000 0X0000 0X0000
DATA T4
% .PRE .ACC %
% T4:0 % 0 2
% T4:1 % 150 0
% T4:2 % 400 0
% T4:3 % 222 82
% T4:4 % 1000 0
% T4:5 % 5 5
% T4:6 % 10 10
% T4:7 % 150 0
% T4:8 % 20 4
% T4:9 % 50 9
% T4:10 % 200 200
% T4:11 % 111 0
% T4:12 % 50 50
% T4:13 % 250 0
% T4:14 % 666 0
% T4:15 % 1000 1003
% T4:16 % 400 0
% T4:17 % 100 63
% T4:18 % 5 0
% T4:19 % 300 0
% T4:20 % 200 0
% T4:21 % 200 0
% T4:22 % 200 0
% T4:23 % 250 0
% T4:24 % 666 0
% T4:25 % 666 0
% T4:26 % 666 0
% T4:27 % 250 0
% T4:28 % 250 0
% T4:29 % 5000 0
% T4:30 % 333 0
% T4:31 % 444 330
% T4:32 % 222 74
% T4:33 % 222 69
% T4:34 % 1111 0
% T4:35 % 23 0
DATA C5
% .PRE .ACC %
% C5:0 % 32766 0
DATA R6
% .LEN .POS %
% R6:0 % 1250 0
% R6:1 % 16 0
% R6:2 % 1050 0
% R6:3 % 1050 0
% R6:4 % 1250 0
% R6:5 % 1250 0
% R6:6 % 1713 0
% R6:7 % 16 0
% R6:8 % 1024 0
% R6:9 % 3 0
% R6:10 % 1713 0
% R6:11 % 1050 0
% R6:12 % 10 0
% R6:13 % 10 0
% R6:14 % 10 0
% R6:15 % 10 0
% R6:16 % 1713 0
% R6:17 % 1713 0
% R6:18 % 1050 0
% R6:19 % 10 0
DATA N7
% N7:0 % -32351 3 870 238 3 0 0 0 500 43
% N7:10 % 1000 43 0 8 22 22 1000 2000 50 1050
% N7:20 % 0 1329 16 2000 0 48 0 0 0 250
% N7:30 % 666 -17477 150 0 728 638 40 11 0 11
% N7:40 % 2 38 1 37 142 1310 5722 1310 0 16
% N7:50 % 15 16 16 16 17 857 100 0 0 3
% N7:60 % 1713 1713 1050 868 1034 1024 4999 5 400 400
% N7:70 % 100 200 300 400 90 190 290 390 10061 -32406
% N7:80 % 0 0 1266 1274 1370 1379 13 10 0 0
% N7:90 % 2011 4 4 12 1 13 10 222 222 12
% N7:100 % 1003 90 110 100 175 25 0 0 0 0
% N7:190 % -128 27477 27605 32767 0 0 0 0 0 0
DATA F8
% F8:0 % 6
DATA L13
% L13:0 % 237384 425175 0 243611 630391
% L13:5 % 1 188142 162 570538 150087
% L13:10 % 158724 -3 0 15 90
% L13:15 % -1463566461 -2147483648 2147483647 2147483647 82058
% L13:20 % 622844517 -950870993 777 -1022733994 100
% L13:25 % 0 -1023197984 0 0 -1557899308
% L13:30 % 94331986 -1022733998 1020000 -1558345713 1444
% L13:35 % 0 0 0 1495855197 1495855229
% L13:40 % 21801 1000000000 1000000 -1558345741 -1557894008
% L13:45 % -1557893964 15 0 28 575851364
% L13:50 % 15244658 162 -1542513552 0 0
% L13:55 % 15244629 78946679 17565 82392473 82399452
% L13:60 % 26974 1935674 0 600 13
% L13:65 % 100 1300 1495819343 1495819405 2
% L13:70 % 579072579 584 8 2180100 575851364
% L13:75 % 14 30 100 -1542514318 -1
% L13:80 % 557730 74 -74 40 1756540
% L13:85 % 274296 281 280 0 15244659
% L13:90 % 15244630 3 284703 5 -1557893981
% L13:95 % 99 229 0 -1557893940 41
% L13:100 % 4100 7 856800 1111 450
% L13:105 % 41 568360 575940102 39 575940097
% L13:110 % 5 55 110 -997781568 -997781574
% L13:115 % -997781568 6 3 -997781571 1000
% L13:120 % 5075 40 165 133 179
% L13:125 % 0 579072579 27400 3276500 274297
% L13:130 % 55 110 0 249 -249
% L13:135 % 0 500 274296 1000 0
% L13:140 % 49 -49 36 50 50
% L13:145 % 163 5 78946782 5 6
% L13:150 % 12 20 43 -43 3
% L13:155 % 100 -10 0 26 4589052
% L13:160 % 5 27 24 1220 45
% L13:165 % -997781178 -997781169 -997781178 -997781169 6707
% L13:170 % 12817 198 198 500 200
% L13:175 % 4 4 524330 536870935 38
% L13:180 % 1495871505 7 50882 1000000 280000000
% L13:185 % 0 0 1495871438 7 50750
% L13:190 % 279000000 67108864 0 0 0
% L13:195 % 0 0 0 0 134217728
% L13:200 % 33554432 0 0 18432 0
% L13:205 % 0 0 0 424319 1496837
% L13:225 % 0 1048576 0 0 0
% L13:230 % 4096 0 0 1024 0
% L13:235 % 0 2097152 0 0 0
% L13:245 % 0 0 0 561152 0
DATA L19
% L19:0 % -1557899095 -1557898888 -1557898669 -1557898460 -1557898244
% L19:5 % -1557898028 -1557897806 -1557897587 -1557897379 -1557897176
% L19:10 % -1557896964 -1557896755 -1557896550 -1557896336 -1557896134
% L19:15 % -1557895940 -1557899308 0 0 0
% L19:25 % 0 0 0 8 33587200
% L19:30 % 131072 0 -2147483648 0 -2147483648
% L19:45 % 256 0 0 0 5250
DATA L20
% L20:0 % -1557896736 -1557896532 -1557896314 -1557896101 -1557895878
% L20:5 % -1557895660 -1557895456 -1557895242 -1557895034 -1557894826
% L20:10 % -1557894618 -1557894409 -1557894206 -1557894008 -1557915064
% L20:15 % -1557914860 -1557914652 -1557914429 -1557914210 -1557914007
% L20:20 % -1557913809 -1557913586 -1557913381 -1557913163 -1557912965
% L20:25 % -1557912771 -1557912554 -1557912349 -1557912121 -1557911928
% L20:30 % -1557911715 -1557911497 -1557911279 -1557911070 -1557910852
% L20:35 % -1557910648 -1557910416 -1557910227 -1557909994 -1557909811
% L20:40 % -1557909597 -1557909374 -1557909156 -1557908948 -1557908749
% L20:45 % -1557908521 -1557908307 -1557908094 -1557907881 -1557907673
% L20:50 % -1557907464 -1557907250 -1557907032 -1557906823 -1557906600
% L20:55 % -1557906397 -1557906184 -1557905990 -1557905772 -1557905574
% L20:60 % -1557905366 -1557905182 -1557904959 -1557904741 -1557904533
% L20:65 % -1557904330 -1557904112 -1557903904 -1557903686 -1557903473
% L20:70 % -1557903260 -1557903048 -1557902839 -1557902621 -1557902424
% L20:75 % -1557902206 -1557901992 -1557901784 -1557901566 -1557901358
% L20:80 % -1557901140 -1557900942 -1557900729 -1557900525 -1557900311
% L20:85 % -1557900094 -1557899678 -1557899459 -1557899266 -1557899042
% L20:90 % -1557898834 -1557898621 -1557898432 -1557898229 -1557898015
% L20:95 % -1557897807 -1557897589 -1557897376 -1557897168 -1557896959
% L20:100 % 0 524288 0 2 0
% L20:105 % 0 1 0 0 0
% L20:120 % 0 0 128 1073741824 0
% L20:125 % 0 0 0 1048576 0
% L20:130 % 1073741824 0 0 0 0
% L20:145 % 0 0 0 0 268435456
% L20:150 % 0 512 0 0 0
% L20:165 % 0 0 1 0 131072
% L20:175 % 0 0 0 0 1048576
% L20:185 % 4194304 0 67108864 0 0
% L20:190 % 0 -2147483648 0 0 0
% L20:195 % 0 0 512 0 268435712
% L20:200 % 0 0 32768 0 0
% L20:210 % 8388608 0 0 0 0
% L20:225 % 16777216 0 0 4194304 0
% L20:235 % 64 68 0 128 0
% L20:240 % 0 0 0 64 0
DATA L21
% L21:0 % -997781728 -997781687 -997781643 -997781600 -997781555
% L21:5 % -997781511 -997781470 -997781427 -997781385 -997781343
% L21:10 % -997781301 -997781259 -997781218 -997781178 -997785424
% L21:15 % -997785383 -997785341 -997785296 -997785252 -997785211
% L21:20 % -997785171 -997785126 -997785085 -997785041 -997785001
% L21:25 % -997784962 -997784918 -997784877 -997784831 -997784792
% L21:30 % -997784749 -997784705 -997784661 -997784619 -997784575
% L21:35 % -997784534 -997784487 -997784449 -997784402 -997784365
% L21:40 % -997784322 -997784277 -997784233 -997784191 -997784151
% L21:45 % -997784105 -997784062 -997784019 -997783976 -997783934
% L21:50 % -997783892 -997783849 -997783805 -997783763 -997783718
% L21:55 % -997783677 -997783634 -997783595 -997783551 -997783511
% L21:60 % -997783469 -997783432 -997783387 -997783343 -997783301
% L21:65 % -997783260 -997783216 -997783174 -997783130 -997783087
% L21:70 % -997783044 -997783001 -997782959 -997782915 -997782875
% L21:75 % -997782831 -997782788 -997782746 -997782702 -997782660
% L21:80 % -997782616 -997782576 -997782533 -997782492 -997782449
% L21:85 % -997782405 -997782321 -997782277 -997782238 -997782193
% L21:90 % -997782151 -997782108 -997782070 -997782029 -997781986
% L21:95 % -997781944 -997781900 -997781857 -997781815 -997781773
% L21:110 % 0 4096 0 0 -2147483648
% L21:115 % 0 0 0 2048 0
% L21:120 % 0 0 262144 0 0
% L21:130 % 0 0 0 8388608 0
% L21:135 % 0 0 0 0 32
% L21:140 % 33554432 0 0 1024 0
% L21:145 % 0 0 0 0 1024
% L21:150 % 0 0 0 0 1073741824
% L21:155 % 0 0 0 0 524288
% L21:165 % 0 0 0 16384 32
% L21:170 % 8192 0 0 0 0
% L21:180 % 0 0 0 0 148
% L21:205 % 0 2048 0 0 0
% L21:210 % 0 0 0 75776 0
% L21:240 % 16 0 0 0 4
% L21:250 % 1024 0 0 0 32
DATA L22
% L22:0 % -1557896056 -1557895833 -1557895615 -1557895411 -1557895198
% L22:5 % -1557894989 -1557894781 -1557894573 -1557894365 -1557894162
% L22:10 % -1557893964 -1557904488 -1557904285 -1557904067 -1557903859
% L22:15 % -1557903642 -1557903429 -1557903216 -1557903003 -1557902795
% L22:20 % -1557902577 -1557902379 -1557902161 -1557901947 -1557901740
% L22:25 % -1557901522 -1557901313 -1557901096 -1557900897 -1557900684
% L22:30 % -1557900480 -1557900267 -1557900049 -1557899633 -1557899415
% L22:35 % -1557899221 -1557898998 -1557898789 -1557898576 -1557898388
% L22:40 % -1557898184 -1557897971 -1557897762 -1557897544 -1557897331
% L22:45 % -1557897123 -1557896915 -1557896691 -1557896488 -1557896269
DATA L23
% L23:0 % -997781591 -997781546 -997781502 -997781461 -997781418
% L23:5 % -997781376 -997781334 -997781292 -997781250 -997781209
% L23:10 % -997781169 -997783292 -997783251 -997783207 -997783165
% L23:15 % -997783121 -997783078 -997783035 -997782992 -997782950
% L23:20 % -997782906 -997782866 -997782822 -997782779 -997782737
% L23:25 % -997782693 -997782651 -997782607 -997782567 -997782524
% L23:30 % -997782483 -997782440 -997782396 -997782312 -997782268
% L23:35 % -997782229 -997782184 -997782142 -997782099 -997782061
% L23:40 % -997782020 -997781977 -997781935 -997781891 -997781848
% L23:45 % -997781806 -997781764 -997781719 -997781678 -997781634
DATA L30
% L30:0 % -1558348352 -1558348094 -1558347861 -1558347613 -1558347386
% L30:5 % -1558347149 -1558346912 -1558346684 -1558346446 -1558346218
% L30:10 % -1558345970 -1558345741 -1612153860 -1611806862 -1611786971
% L30:15 % -1611757888 -1558423573 -1558423341 -1558423112 -1558422874
% L30:20 % -1558422651 -1558356915 -1558356677 -1558356455 -1558356217
% L30:25 % -1558355979 -1558355745 -1558355512 -1558355273 -1558355021
% L30:30 % -1558354786 -1558354544 -1558354301 -1558354063 -1558353824
% L30:35 % -1558353581 -1558353354 -1558353125 -1558352902 -1558352674
% L30:40 % -1558352441 -1558350432 -1558350197 -1558349970 -1558349747
% L30:45 % -1558349510 -1558349281 -1558349033 -1558348799 -1558348571
DATA L31
% L31:0 % 575850837 575850889 575850936 575850986 575851032
% L31:5 % 575851080 575851128 575851174 575851222 575851268
% L31:10 % 575851318 575851364 564997934 565073008 565077019
% L31:15 % 565082883 575835671 575835718 575835764 575835812
% L31:20 % 575835857 575849111 575849159 575849204 575849252
% L31:25 % 575849300 575849347 575849394 575849442 575849493
% L31:30 % 575849540 575849589 575849638 575849686 575849734
% L31:35 % 575849783 575849829 575849875 575849920 575849966
% L31:40 % 575850013 575850418 575850465 575850511 575850556
% L31:45 % 575850604 575850650 575850700 575850747 575850793
DATA L32
% L32:0 % -1542513552 -1542513102 -1542514004 -1557910109 -1557909896
% L32:5 % -1557909688 -1557909474 -1557909271 -1557909056 -1557908847
% L32:10 % -1557908633 -1557908424 -1557908211 -1557907997 -1557907785
% L32:15 % -1557907586 -1557907374 -1557907159 -1557906946 -1557906759
% L32:20 % -1557906550 -1557906338 -1557906134 -1557905911 -1557905708
% L32:25 % -1557905494 -1557905285 -1557905066 -1557904859 -1557904640
% L32:30 % -1557904432 -1557904209 -1557903991 -1557903783 -1557903579
% L32:35 % -1557903367 -1557903159 -1557902951 -1557902743 -1557902539
% L32:40 % -1557902347 -1542622975 -1542622525 -1557912231 -1557912018
% L32:45 % -1557911805 -1557911591 -1557911383 -1557911170 -1557910951
DATA L33
% L33:0 % 579073328 579073578 579073077 575939187 575939230
% L33:5 % 575939272 575939315 575939356 575939399 575939441
% L33:10 % 575939484 575939526 575939569 575939612 575939655
% L33:15 % 575939695 575939738 575939781 575939824 575939862
% L33:20 % 575939904 575939947 575939988 575940033 575940074
% L33:25 % 575940117 575940159 575940203 575940245 575940289
% L33:30 % 575940331 575940376 575940420 575940462 575940503
% L33:35 % 575940546 575940588 575940630 575940672 575940713
% L33:40 % 575940752 579017052 579017281 575938759 575938802
% L33:45 % 575938845 575938888 575938930 575938973 575939017
DATA B34
% B34:110 % 0X0000 0X0000 0X0000 0X0000 0X0000 0X0000 0X0200 0X0000 0X0000 0X0000
% B34:120 % 0X0000 0X0000 0X0000 0X0000 0X0000 0X0000 0X0000 0X8000
DATA B35
% B35:110 % 0X0000 0X0000 0X0200 0X0000 0X0000 0X0000 0X0000 0X0000 0X0000 0X0000
DATA B37
% B37:0 % 0X0000 0X0000 0X2000 0X0000 0X0000 0X0000 0X0000 0X0000 0X0000 0X0000
DATA B40
% B40:0 % 0XAAAA
DATA B100
% B100:0 % 0X2F00 0X80A0 0X0004 0X0000 0X0000 0X0000 0X0000 0X0000 0X0000 0X0000
DATA N101
% N101:0 % 128 647 0 0 1182 105 867 1200 1200 1260
% N101:10 % 1269 1616 10 19004 1187 0 3050 222 333 444
% N101:20 % 1000 500 400 0 0 0 222 222 0 0
DATA L102
% L102:0 % 50 10 5510 5502 5500
% L102:5 % 5500 0 0 0 0
% L102:10 % 0 3798 0 0 284703
% L102:15 % 0 30 10 30 10
% L102:20 % 42 5 0 3 27
% L102:25 % 28 18 41 0 18
% L102:30 % 584 8 8568 0 1904
% L102:35 % 149 1200 0 999999 24
% L102:40 % 90 2 0 1 0
